// TIA Portal V16 export
// export: Created 2022-08-08T12:29:17.9300338Z, ExportSetting WithDefaults, DisplayName Totally Integrated Automation Portal, DisplayVersion V16, DisplayName TIA Portal Version Control Interface, DisplayVersion V16, DisplayName TIA Portal Openness, DisplayVersion V16, DisplayName SINAMICS Startdrive Advanced, DisplayVersion V16, DisplayName SINAMICS Startdrive G130, G150, S120, S150, SINAMICS MV, S210, DisplayVersion V16, DisplayName SINAMICS Startdrive G110M, G120, G120C, G120D, G120P, DisplayVersion V16, DisplayName STEP 7 Professional, DisplayVersion V16, DisplayName STEP 7 Safety, DisplayVersion V16, DisplayName WinCC Professional, DisplayVersion V16
ORGANIZATION_BLOCK "Automatic_Gate_Example"   // OB1, LAD, ProgramCycle
TITLE = "Main Program Sweep (Cycle)"
{ S7_Optimized_Access := 'TRUE' }
VERSION : 0.1
// stored: AutoNumber true, IsIECCheckEnabled false, SetENOAutomatically false
   VAR_INPUT
      Initial_Call : Bool;   // Initial call of this OB
      Remanence : Bool;   // =True, if remanent data are available
   END_VAR
BEGIN

REGION Network 1
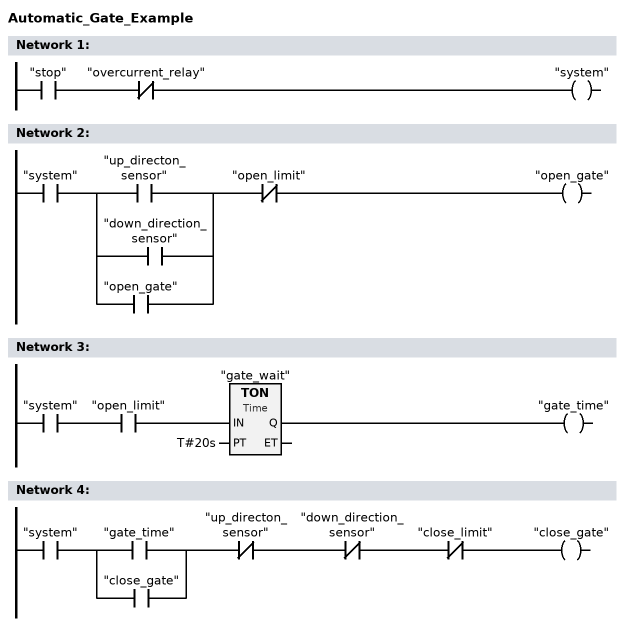
   RUNG wire#powerrail
      Contact( "stop" )
      I_Contact( "overcurrent_relay" )
      Coil( "system" )
   END_RUNG
   // the same network as SCL:
   "system" := "stop" AND NOT "overcurrent_relay";
END_REGION

REGION Network 2
   RUNG wire#powerrail
      Contact( "system" )
      wire#w1
      Contact( "up_directon_sensor" )
      wire#w2
      I_Contact( "open_limit" )
      Coil( "open_gate" )
   END_RUNG
   RUNG wire#w1
      Contact( "down_direction_sensor" )
   END_RUNG wire#w2
   RUNG wire#w1
      Contact( "open_gate" )
   END_RUNG wire#w2
   // the same network as SCL:
   "open_gate" := "system" AND ("up_directon_sensor" OR "down_direction_sensor" OR "open_gate") AND NOT "open_limit";
END_REGION

REGION Network 3
   RUNG wire#powerrail
      Contact( "system" )
      Contact( "open_limit" )
      { S7_Templates := "time_type := Time" } "gate_wait".TON(pt := T#20s, et =>)
      Coil( "gate_time" )
   END_RUNG
   // the same network as SCL:
   "gate_wait".TON(IN := "system" AND "open_limit", PT := T#20s);
   "gate_time" := "gate_wait".Q;
END_REGION

REGION Network 4
   RUNG wire#powerrail
      Contact( "system" )
      wire#w1
      Contact( "gate_time" )
      wire#w2
      I_Contact( "up_directon_sensor" )
      I_Contact( "down_direction_sensor" )
      I_Contact( "close_limit" )
      Coil( "close_gate" )
   END_RUNG
   RUNG wire#w1
      Contact( "close_gate" )
   END_RUNG wire#w2
   // the same network as SCL:
   "close_gate" := "system" AND ("gate_time" OR "close_gate") AND NOT "up_directon_sensor" AND NOT "down_direction_sensor" AND NOT "close_limit";
END_REGION
END_ORGANIZATION_BLOCK
